// TIA Portal V16 export
// export: Created 2022-02-04T14:40:23.4312381Z, ExportSetting WithDefaults, DisplayName Totally Integrated Automation Portal, DisplayVersion V16 Update 1, DisplayName TIA Portal Version Control Interface, DisplayVersion V16, DisplayName TIA Portal Openness, DisplayVersion V16, DisplayName SINAMICS Startdrive Advanced, DisplayVersion V16 Update 5, DisplayName SINAMICS Startdrive G130, G150, S120, S150, SINAMICS MV, S210, DisplayVersion V16 Update 5, DisplayName SINAMICS Startdrive G110M, G120, G120C, G120D, G120P, G115D, DisplayVersion V16 Update 5, DisplayName STEP 7 Professional, DisplayVersion V16, DisplayName STEP 7 Safety, DisplayVersion V16, DisplayName WinCC Advanced, DisplayVersion V16, DisplayName SIMATIC Visualization Architect, DisplayVersion V16
DATA_BLOCK "KeyFazer_CNTL_DB"   // DB28
AUTHOR : Aspir
VERSION : 0.1
// stored: AutoNumber true, InstanceOfName KeyFazer_CNTL, InstanceOfType FB
"KeyFazer_CNTL"
   // VAR_INPUT
   //    keyfazer_1 : Bool;
   //    keyfazer_2 : Bool;
   //    enableSensors : Bool;
   // END_VAR
   // VAR_OUTPUT
   //    WheelChanged : Bool;
   //    ActualWheelSig : Bool;
   //    Chain : Bool;
   //    Window : Bool;
   //    FaultKeyFazer : Bool;
   // END_VAR
   // VAR RETAIN
   //    active_wheel : Bool;
   //    validSig_old : Bool;
   //    changing_wheel : Bool;
   //    memento_act_wheel : Bool;
   //    real_chain : Bool;
   //    AntiNoValidFront_timer : TON;
   // END_VAR
BEGIN
END_DATA_BLOCK
